{attribute 'GeneratedUsingTerminal: EP1122-0001-0016'}
{attribute addProperty BoxType "EP1122-0001-0016"}
{attribute addProperty Id "A_0025_EP1122_0001_0017A_0025_EP1122_0001_0017_880ECFB91450"}
{attribute addProperty CRC "121032131"}
{attribute addProperty Size "1450"}
TYPE A_0024_EP1122_0001_0016_0736CDC3 EXTENDS EP1122_AB5A9467 :
STRUCT
	{attribute addProperty Name "A_0025_EP1122_0001_0017"}
	{attribute addProperty PreviousPort "A_0024(EP1122-0001-0016) : D"}
	A_0025_EP1122_0001_0017 : A_0025_EP1122_0001_0017_880ECFB9;
END_STRUCT
END_TYPE

(* stored: Version 1.2.0.0, ProductVersion 3.1.4024.9
   DUT A_0024_EP1122_0001_0016_0736CDC3: Id {6e8cb7a0-faa4-4183-9b3c-36d0586b8d58} *)
